        // ===========================================
        // STEP 549: PressShaftPutProcessFinish
        // ===========================================
        STEP_ST10_Flow5_FRobot_1_PressShaftPutProcessFinish:
            // Action Qualifier=S
            // Token: #ioPM_Inface.ProcessComplete
            #ioPM_Inface.ProcessComplete := TRUE;
            // Action Qualifier=R
            // Token: #ioPM_Inface.ProcessStart
            #ioPM_Inface.ProcessStart := FALSE;
            // Action Qualifier=N
            // Token: "AutoProcessData".F_Robot1Grip1.PartStatus := 0
            "AutoProcessData".F_Robot1Grip1.PartStatus := 0;

            // Transition to next step: 355
            IF TRUE THEN  // Sequential transition - review XML for actual condition
                #State := STEP_ST10_Flow5_FRobot_1_StartRobotScanRing;
            END_IF;

        // ===========================================
        // STEP 355: StartRobotScanRing
        // ===========================================
        STEP_ST10_Flow5_FRobot_1_StartRobotScanRing:
            // Action Qualifier=N
            // Token: "KukaRobot1_CtrlDB".sPLCtoROB.User.Cycle.DI261_RingScanReq
            "KukaRobot1_CtrlDB".sPLCtoROB.User.Cycle.DI261_RingScanReq;

            // Transition to next step: 382
            IF TRUE THEN  // Sequential transition - review XML for actual condition
                #State := STEP_ST10_Flow5_FRobot_1_RobotManuallyMoved_;
            END_IF;

        // ===========================================
        // STEP 382: RobotManuallyMoved?
        // ===========================================
        STEP_ST10_Flow5_FRobot_1_RobotManuallyMoved_:
            // No actions in XML

            // Transition to next step: 335
            IF TRUE THEN  // Sequential transition - review XML for actual condition
                #State := STEP_ST10_Flow5_FRobot_1_RobotScanGripperReachPos1;
            END_IF;

        // ===========================================
        // STEP 335: RobotScanGripperReachPos1
        // ===========================================
        STEP_ST10_Flow5_FRobot_1_RobotScanGripperReachPos1:
            // No actions in XML

            // Transition to next step: 267
            IF TRUE THEN  // Sequential transition - review XML for actual condition
                #State := STEP_ST10_Flow5_FRobot_1_Data_Clear_7;
            END_IF;

        // ===========================================
        // STEP 267: Data Clear_7
        // ===========================================
        STEP_ST10_Flow5_FRobot_1_Data_Clear_7:
            // Action Qualifier=N, Event="S1"
            // Token: "AutoProcessData".F_Robot1Grip1 := "AutoProcessData".ClearData
            "AutoProcessData".F_Robot1Grip1 := "AutoProcessData".ClearData;

            // Transition to next step: 245
            IF TRUE THEN  // Sequential transition - review XML for actual condition
                #State := STEP_ST10_Flow5_FRobot_1_CheckScanReady;
            END_IF;

        // ===========================================
        // STEP 245: CheckScanReady
        // ===========================================
        STEP_ST10_Flow5_FRobot_1_CheckScanReady:
            // No actions in XML

            // Transition to next step: 133
            IF TRUE THEN  // Sequential transition - review XML for actual condition
                #State := STEP_ST10_Flow5_FRobot_1_Brake_Test;
            END_IF;

        // ===========================================
        // STEP 133: Brake_Test
        // ===========================================
        STEP_ST10_Flow5_FRobot_1_Brake_Test:
            // Action Qualifier=R
            // Token: #ioPM_Inface.ProcessComplete
            #ioPM_Inface.ProcessComplete := FALSE;
            // Action Qualifier=S
            // Token: #ioPM_Inface.ProcessStart
            #ioPM_Inface.ProcessStart := TRUE;

            // Transition to next step: 701
            IF TRUE THEN  // Sequential transition - review XML for actual condition
                #State := STEP_ST10_Flow5_FRobot_1_ReqRobotToMantenPos;
            END_IF;

        // ===========================================
        // STEP 701: ReqRobotToMantenPos
        // ===========================================
        STEP_ST10_Flow5_FRobot_1_ReqRobotToMantenPos:
            // Action Qualifier=N
            // Token: "KukaRobot1_CtrlDB".sPLCtoROB.User.Cycle.DI297_MaintainRequest
            "KukaRobot1_CtrlDB".sPLCtoROB.User.Cycle.DI297_MaintainRequest;

            // Transition to next step: 849
            IF TRUE THEN  // Sequential transition - review XML for actual condition
                #State := STEP_ST10_Flow5_FRobot_1_NG3_PutProcessFinish;
            END_IF;

        // ===========================================
        // STEP 849: NG3 PutProcessFinish
        // ===========================================
        STEP_ST10_Flow5_FRobot_1_NG3_PutProcessFinish:
            // Action Qualifier=S
            // Token: #ioPM_Inface.ProcessComplete
            #ioPM_Inface.ProcessComplete := TRUE;
            // Action Qualifier=R
            // Token: #ioPM_Inface.ProcessStart
            #ioPM_Inface.ProcessStart := FALSE;

            // Transition to next step: 800
            IF TRUE THEN  // Sequential transition - review XML for actual condition
                #State := STEP_ST10_Flow5_FRobot_1_NG_3_PutProcess;
            END_IF;

        // ===========================================
        // STEP 800: NG 3 PutProcess
        // ===========================================
        STEP_ST10_Flow5_FRobot_1_NG_3_PutProcess:
            // No actions in XML

            // Transition to next step: 242
            IF TRUE THEN  // Sequential transition - review XML for actual condition
                #State := STEP_ST10_Flow5_FRobot_1_Wait_ScanFinish;
            END_IF;

        // ===========================================
        // STEP 242: Wait ScanFinish
        // ===========================================
        STEP_ST10_Flow5_FRobot_1_Wait_ScanFinish:
            // No actions in XML

            // Transition to next step: 309
            IF TRUE THEN  // Sequential transition - review XML for actual condition
                #State := STEP_ST10_Flow5_FRobot_1_WaitRobotReachPos1;
            END_IF;

        // ===========================================
        // STEP 309: WaitRobotReachPos1
        // ===========================================
        STEP_ST10_Flow5_FRobot_1_WaitRobotReachPos1:
            // No actions in XML

            // Transition to next step: 347
            IF TRUE THEN  // Sequential transition - review XML for actual condition
                #State := STEP_ST10_Flow5_FRobot_1_WaitRobotGripHaveStatus_1;
            END_IF;

        // ===========================================
        // STEP 347: WaitRobotGripHaveStatus_1
        // ===========================================
        STEP_ST10_Flow5_FRobot_1_WaitRobotGripHaveStatus_1:
            // No actions in XML

            // Transition to next step: 260
            IF TRUE THEN  // Sequential transition - review XML for actual condition
                #State := STEP_ST10_Flow5_FRobot_1_DataMove_3;
            END_IF;

        // ===========================================
        // STEP 260: DataMove_3
        // ===========================================
        STEP_ST10_Flow5_FRobot_1_DataMove_3:
            // Action Qualifier=N, Event="S1"
            // Token: "AutoProcessData".B_Press1.RingCode_1 := "AutoProcessData".F_Robot1Grip2.RingCode_1
            "AutoProcessData".B_Press1.RingCode_1 := "AutoProcessData".F_Robot1Grip2.RingCode_1;
            // Action Qualifier=N, Event="S1"
            // Token: "AutoProcessData".F_Robot1Grip2 := "AutoProcessData".ClearData
            "AutoProcessData".F_Robot1Grip2 := "AutoProcessData".ClearData;
            // Action Qualifier=N
            // Token: "AutoProcessData".B_Press1.PartStatus := 220
            "AutoProcessData".B_Press1.PartStatus := 220;

            // Transition to next step: 919
            IF TRUE THEN  // Sequential transition - review XML for actual condition
                #State := STEP_ST10_Flow5_FRobot_1_MasteringTestFinish;
            END_IF;

        // ===========================================
        // STEP 919: MasteringTestFinish
        // ===========================================
        STEP_ST10_Flow5_FRobot_1_MasteringTestFinish:
            // Action Qualifier=R
            // Token: "Robot_DB".Robot_1.MasteringTest_Req
            "Robot_DB".Robot_1.MasteringTest_Req := FALSE;

            // Transition to next step: 326
            IF TRUE THEN  // Sequential transition - review XML for actual condition
                #State := STEP_ST10_Flow5_FRobot_1_StartRobotPickPalletShaft;
            END_IF;

        // ===========================================
        // STEP 326: StartRobotPickPalletShaft
        // ===========================================
        STEP_ST10_Flow5_FRobot_1_StartRobotPickPalletShaft:
            // Action Qualifier=N
            // Token: "KukaRobot1_CtrlDB".sPLCtoROB.User.Cycle.DI241_PickShaftPalletReq
            "KukaRobot1_CtrlDB".sPLCtoROB.User.Cycle.DI241_PickShaftPalletReq;

            // Transition to next step: 130
            IF TRUE THEN  // Sequential transition - review XML for actual condition
                #State := STEP_ST10_Flow5_FRobot_1_PickTable;
            END_IF;

        // ===========================================
        // STEP 130: PickTable
        // ===========================================
        STEP_ST10_Flow5_FRobot_1_PickTable:
            // Action Qualifier=R
            // Token: #ioPM_Inface.ProcessComplete
            #ioPM_Inface.ProcessComplete := FALSE;
            // Action Qualifier=S
            // Token: #ioPM_Inface.ProcessStart
            #ioPM_Inface.ProcessStart := TRUE;

            // Transition to next step: 368
            IF TRUE THEN  // Sequential transition - review XML for actual condition
                #State := STEP_ST10_Flow5_FRobot_1_WaitRobotFinish_8;
            END_IF;

        // ===========================================
        // STEP 368: WaitRobotFinish_8
        // ===========================================
        STEP_ST10_Flow5_FRobot_1_WaitRobotFinish_8:
            // No actions in XML

            // Transition to next step: 331
            IF TRUE THEN  // Sequential transition - review XML for actual condition
                #State := STEP_ST10_Flow5_FRobot_1_Gripe1StatusAlarm;
            END_IF;

        // ===========================================
        // STEP 331: Gripe1StatusAlarm
        // ===========================================
        STEP_ST10_Flow5_FRobot_1_Gripe1StatusAlarm:
            // Action Qualifier=S
            // Token: "ST10_DeviceError".F.Robot_1.Grip1Error
            "ST10_DeviceError".F.Robot_1.Grip1Error := TRUE;

            // Transition to next step: 248
            IF TRUE THEN  // Sequential transition - review XML for actual condition
                #State := STEP_ST10_Flow5_FRobot_1_CodeMove;
            END_IF;

        // ===========================================
        // STEP 248: CodeMove
        // ===========================================
        STEP_ST10_Flow5_FRobot_1_CodeMove:
            // Action Qualifier=N
            // Token: "AutoProcessData".F_Robot1Grip2.RingCode_1 := "KeyenceSR1000Ctrl_804A1DB".sHMI.Status.CurrentCode
            "AutoProcessData".F_Robot1Grip2.RingCode_1 := "KeyenceSR1000Ctrl_804A1DB".sHMI.Status.CurrentCode;

            // Transition to next step: 315
            IF TRUE THEN  // Sequential transition - review XML for actual condition
                #State := STEP_ST10_Flow5_FRobot_1_WaitPos3ScanFinish;
            END_IF;

        // ===========================================
        // STEP 315: WaitPos3ScanFinish
        // ===========================================
        STEP_ST10_Flow5_FRobot_1_WaitPos3ScanFinish:
            // No actions in XML

            // Transition to next step: 365
            IF TRUE THEN  // Sequential transition - review XML for actual condition
                #State := STEP_ST10_Flow5_FRobot_1_WaitRobotFinish_7;
            END_IF;

        // ===========================================
        // STEP 365: WaitRobotFinish_7
        // ===========================================
        STEP_ST10_Flow5_FRobot_1_WaitRobotFinish_7:
            // No actions in XML

    END_CASE;

    // UPDATE ioPM_Inface
    #ioPM_Inface.InitialRun := #act_InitialRun;
    #ioPM_Inface.InitialOK := #act_InitialOK;
    #ioPM_Inface.WaitRunning := #act_WaitRunning;
    #ioPM_Inface.Running := #act_Running;
    #ioPM_Inface.ProcessComplete := #act_ProcessComplete;
    #ioPM_Inface.ProcessStart := #act_ProcessStart;
    #ioPM_Inface.UnPause := #act_UnPause;

    // ERROR HANDLING
    IF #bError THEN
        #ioStatus := 900;
        #oAlarmID := INT_TO_WORD(#wErrorID);
    ELSE
        #ioStatus := 0;
        #oAlarmID := 0;
    END_IF;
END_FUNCTION_BLOCK

//=============================================================================
// END OF FILE
//=============================================================================
